Staubli VAL3: onEnterEvent.pgx

program onEnterEvent(string x_sId, bool& x_bSave[])
  local bool l_bFound
  local num l_nX
  local num l_nY
  local string l_sString
  local string l_sMessage
  local bool l_bOk
  local num l_nValue
  local string l_sName
begin
  //
  // NB sEvent is the selected
  // element in the LIST
  //
  l_nX=40-use:nBottomX+find(sEvent,"{")
  // select
  switch nViewMode
    case 0
      // OUT
      call out:getItem(l_sString,x_sId)
    break
    case 1
      // IN
      call in:getItem(l_sString,x_sId)
    break
    case 2
      // COUNT
      call saveInOut:getItem_num(l_sString,x_sId)
    break
  endSwitch
  // set the list
  l_nY=nView+1
  if nViewMode!=2
    // clean the line
    call use:listcursor(use:nView,false)
  endIf
  // read the name
  l_sName=l_sString
  call use:read(l_nX,l_nY,l_sString,14,false)
  // check if already exist
  if !use:bUseEscape and l_sString!=l_sName and l_sString!=""
    switch nViewMode
      case 0
        // OUT
        call out:setItem(l_sString,x_sId)
      break
      case 1
        // IN
        call in:setItem(l_sString,x_sId)
      break
      case 2
        // COUNT
        call NUM:set(l_sString,x_sId)
      break
    endSwitch
    // save it
    x_bSave=true
  endIf
end
